// TIA Portal V19 export
TYPE "IFM_PI1714_IO"
   STRUCT
      Addr : Int;   // IO Address
      Value_p : Real;   // Pressure_Bar
      Value_t : Real;   // Temperature_C
      DeviceStatus : Byte;   // Device Status
      OUT2 : Bool;   // Out 2
      OUT1 : Bool;   // Out 1
      O_DI4 : Bool;   // Port pin 4
      O_DI2 : Bool;   // Port pin 2
      O_DA : Bool;   // Device Attached
      O_DE : Bool;   // Device Error
      O_PQ : Bool;   // Value Valid
   END_STRUCT;
END_TYPE
